(* Logix 5000 project; controller R1USB70001_CWRU_GRID_20120217 vendor 1 type 14 code 54 rev 19.11; software revision 19.01; part 3 of 3 *)
(* tags used below, declared in another part *)
   BAT_AC_VOLTAGE : REAL;
   BAT_AC_VOLTAGE_RAW : REAL;
   BAT_CHARGE_AC_CURRENT : REAL;
   BAT_CHARGE_AC_CURRENT_RAW : REAL;
   BAT_CHARGE_DC_CURRENT : REAL;
   BAT_CHARGE_DC_CURRENT_RAW : REAL;
   BAT_SRC_AC_CURRENT1 : REAL;
   BAT_SRC_AC_CURRENT1_RAW : REAL;
   BAT_SRC_AC_CURRENT2 : REAL;
   BAT_SRC_AC_CURRENT2_RAW : REAL;
   BAT_SRC_DC_CURRENT : REAL;
   BAT_SRC_DC_CURRENT_RAW : REAL;
   CAES_CHARGE_CURRENT : REAL;
   CAES_CHARGE_CURRENT_RAW : REAL;
   CAES_SRC_CURRENT : REAL;
   CAES_SRC_CURRENT_RAW : REAL;
   CAP_MAIN_CURRENT : REAL;
   CAP_MAIN_CURRENT_RAW : REAL;
   COM_TO_GRID_CURRENT : REAL;
   COM_TO_GRID_CURRENT_RAW : REAL;
   CURRENT_SCALE_HIGH : REAL;
   CURRENT_SCALE_LOW : REAL;
   IND_TO_GRID_CURRENT : REAL;
   IND_TO_GRID_CURRENT_RAW : REAL;
   MAINS_AC_VOLTAGE : REAL;
   MAINS_AC_VOLTAGE_RAW : REAL;
   RES_TO_GRID_CURRENT : REAL;
   RES_TO_GRID_CURRENT_RAW : REAL;
   SC_TO_BAT_CURRENT : REAL;
   SC_TO_BAT_CURRENT_RAW : REAL;
   SC_TO_COM_CURRENT : REAL;
   SC_TO_COM_CURRENT_RAW : REAL;
   SC_TO_GRID_CURRENT : REAL;
   SC_TO_GRID_CURRENT_RAW : REAL;
   SC_TO_IND_CURRENT : REAL;
   SC_TO_IND_CURRENT_RAW : REAL;
   SC_TO_RES_CURRENT : REAL;
   SC_TO_RES_CURRENT_RAW : REAL;
   SF_TO_BAT_CURRENT : REAL;
   SF_TO_BAT_CURRENT_RAW : REAL;
   SF_TO_COM_CURRENT : REAL;
   SF_TO_COM_CURRENT_RAW : REAL;
   SF_TO_GRID_CURRENT : REAL;
   SF_TO_GRID_CURRENT_RAW : REAL;
   SF_TO_IND_CURRENT : REAL;
   SF_TO_IND_CURRENT_RAW : REAL;
   SF_TO_RES_CURRENT : REAL;
   SF_TO_RES_CURRENT_RAW : REAL;
   VOLTAGE_SCALE : REAL;
   WF_TO_BAT_CURRENT : REAL;
   WF_TO_BAT_CURRENT_RAW : REAL;
   WF_TO_COM_CURRENT : REAL;
   WF_TO_COM_CURRENT_RAW : REAL;
   WF_TO_GRID_CURRENT : REAL;
   WF_TO_GRID_CURRENT_RAW : REAL;
   WF_TO_IND_CURRENT : REAL;
   WF_TO_IND_CURRENT_RAW : REAL;
   WF_TO_RES_CURRENT : REAL;
   WF_TO_RES_CURRENT_RAW : REAL;
   WT_TO_BAT_CURRENT : REAL;
   WT_TO_BAT_CURRENT_RAW : REAL;
   WT_TO_COM_CURRENT : REAL;
   WT_TO_COM_CURRENT_RAW : REAL;
   WT_TO_GRID_CURRENT : REAL;
   WT_TO_GRID_CURRENT_RAW : REAL;
   WT_TO_IND_CURRENT : REAL;
   WT_TO_IND_CURRENT_RAW : REAL;
   WT_TO_RES_CURRENT : REAL;
   WT_TO_RES_CURRENT_RAW : REAL;
   AP_GP_CH_ACAM : ALIAS FOR ACNR_GP_SC_N2:1:I.Ch1Data;
   AP_GP_SR_ACAM : ALIAS FOR ACNR_GP_SC_N2:1:I.Ch0Data;
   AP_GP_SR_ACVT : ALIAS FOR ACNR_GP_SC_N2:9:I.Ch1Data;
   BT_GP_L1_ACAM1 : ALIAS FOR ACNR_GP_SC_N2:1:I.Ch2Data;
   BT_GP_L1_ACAM2 : ALIAS FOR ACNR_GP_SC_N2:1:I.Ch3Data;
   BT_GP_L1_DCAM : ALIAS FOR ACNR_GP_SC_N2:2:I.Ch2Data;
   BT_GP_L2_ACAM1 : ALIAS FOR ACNR_GP_SC_N2:2:I.Ch0Data;
   BT_GP_L2_DCAM : ALIAS FOR ACNR_GP_SC_N2:2:I.Ch3Data;
   BT_GP_ML_ACVT : ALIAS FOR ACNR_GP_SC_N2:9:I.Ch2Data;
   CB_GP_ML_ACAM : ALIAS FOR ACNR_GP_SC_N2:9:I.Ch0Data;
   CL_GP_GD_ACAM : ALIAS FOR ACNR_GP_SC_N2:5:I.Ch2Data;
   CL_GP_SC_ACAM : ALIAS FOR ACNR_GP_SC_N2:4:I.Ch2Data;
   CL_GP_SF_ACAM : ALIAS FOR ACNR_GP_SC_N2:4:I.Ch3Data;
   CL_GP_WF_ACAM : ALIAS FOR ACNR_GP_SC_N2:5:I.Ch1Data;
   CL_GP_WT_ACAM : ALIAS FOR ACNR_GP_SC_N2:5:I.Ch0Data;
   Comment : DINT[2];
   IL_GP_GD_ACAM : ALIAS FOR ACNR_GP_SC_N2:6:I.Ch3Data;
   IL_GP_SC_ACAM : ALIAS FOR ACNR_GP_SC_N2:5:I.Ch3Data;
   IL_GP_SF_ACAM : ALIAS FOR ACNR_GP_SC_N2:6:I.Ch0Data;
   IL_GP_WF_ACAM : ALIAS FOR ACNR_GP_SC_N2:6:I.Ch2Data;
   IL_GP_WT_ACAM : ALIAS FOR ACNR_GP_SC_N2:6:I.Ch1Data;
   RL_GP_GD_ACAM : ALIAS FOR ACNR_GP_SC_N2:4:I.Ch1Data;
   RL_GP_SC_ACAM : ALIAS FOR ACNR_GP_SC_N2:3:I.Ch0Data;
   RL_GP_SF_ACAM : ALIAS FOR ACNR_GP_SC_N2:3:I.Ch1Data;
   RL_GP_WF_ACAM : ALIAS FOR ACNR_GP_SC_N2:4:I.Ch0Data;
   RL_GP_WT_ACAM : ALIAS FOR ACNR_GP_SC_N2:3:I.Ch2Data;
   SC_GP_BT_ACAM : ALIAS FOR ACNR_GP_SC_N2:8:I.Ch3Data;
   SC_GP_GD_ACAM : ALIAS FOR ACNR_GP_SC_N2:8:I.Ch2Data;
   SF_GP_BT_ACAM : ALIAS FOR ACNR_GP_SC_N2:8:I.Ch1Data;
   SF_GP_GD_ACAM : ALIAS FOR ACNR_GP_SC_N2:8:I.Ch0Data;
   WF_GP_BT_ACAM : ALIAS FOR ACNR_GP_SC_N2:7:I.Ch1Data;
   WF_GP_GD_ACAM : ALIAS FOR ACNR_GP_SC_N2:7:I.Ch0Data;
   WT_GP_BT_ACAM : ALIAS FOR ACNR_GP_SC_N2:7:I.Ch3Data;
   WT_GP_GD_ACAM : ALIAS FOR ACNR_GP_SC_N2:7:I.Ch2Data;
(* MainProgram, continued *)

ROUTINE IMPORT_DATA   (* ladder *)
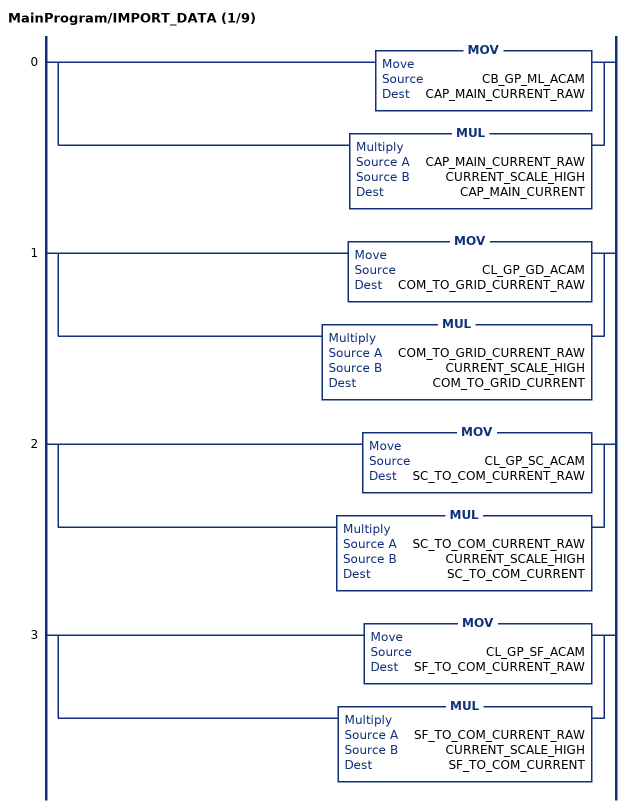
   0: [MOV(CB_GP_ML_ACAM,CAP_MAIN_CURRENT_RAW) ,MUL(CAP_MAIN_CURRENT_RAW,CURRENT_SCALE_HIGH,CAP_MAIN_CURRENT) ];
   1: [MOV(CL_GP_GD_ACAM,COM_TO_GRID_CURRENT_RAW) ,MUL(COM_TO_GRID_CURRENT_RAW,CURRENT_SCALE_HIGH,COM_TO_GRID_CURRENT) ];
   2: [MOV(CL_GP_SC_ACAM,SC_TO_COM_CURRENT_RAW) ,MUL(SC_TO_COM_CURRENT_RAW,CURRENT_SCALE_HIGH,SC_TO_COM_CURRENT) ];
   3: [MOV(CL_GP_SF_ACAM,SF_TO_COM_CURRENT_RAW) ,MUL(SF_TO_COM_CURRENT_RAW,CURRENT_SCALE_HIGH,SF_TO_COM_CURRENT) ];
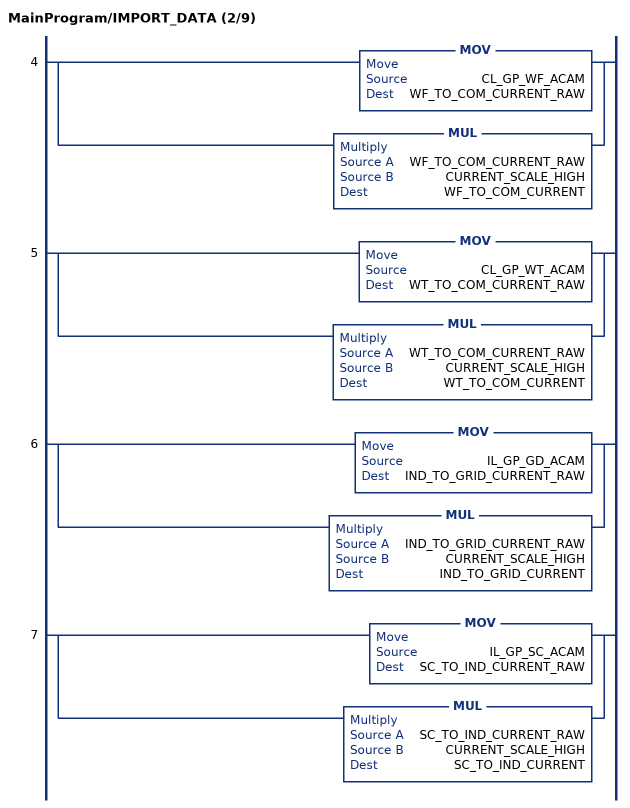
   4: [MOV(CL_GP_WF_ACAM,WF_TO_COM_CURRENT_RAW) ,MUL(WF_TO_COM_CURRENT_RAW,CURRENT_SCALE_HIGH,WF_TO_COM_CURRENT) ];
   5: [MOV(CL_GP_WT_ACAM,WT_TO_COM_CURRENT_RAW) ,MUL(WT_TO_COM_CURRENT_RAW,CURRENT_SCALE_HIGH,WT_TO_COM_CURRENT) ];
   6: [MOV(IL_GP_GD_ACAM,IND_TO_GRID_CURRENT_RAW) ,MUL(IND_TO_GRID_CURRENT_RAW,CURRENT_SCALE_HIGH,IND_TO_GRID_CURRENT) ];
   7: [MOV(IL_GP_SC_ACAM,SC_TO_IND_CURRENT_RAW) ,MUL(SC_TO_IND_CURRENT_RAW,CURRENT_SCALE_HIGH,SC_TO_IND_CURRENT) ];
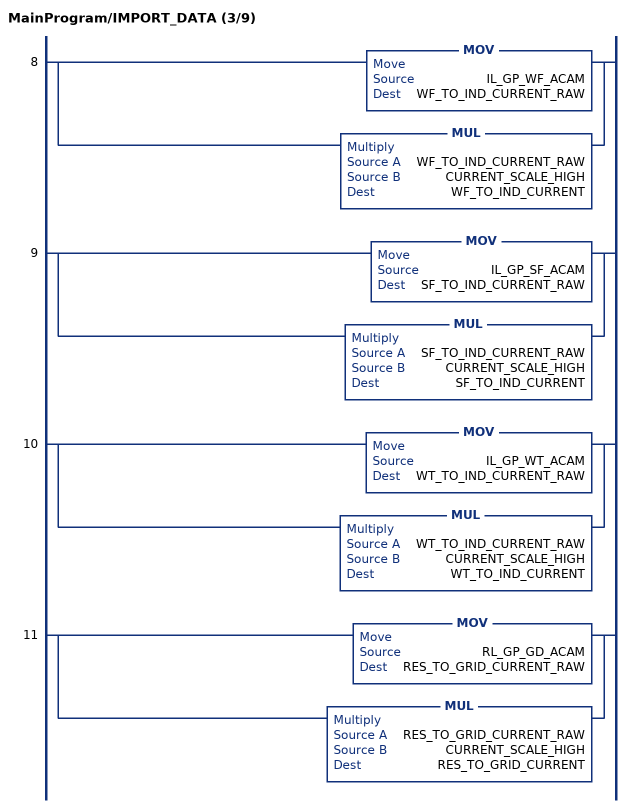
   8: [MOV(IL_GP_WF_ACAM,WF_TO_IND_CURRENT_RAW) ,MUL(WF_TO_IND_CURRENT_RAW,CURRENT_SCALE_HIGH,WF_TO_IND_CURRENT) ];
   9: [MOV(IL_GP_SF_ACAM,SF_TO_IND_CURRENT_RAW) ,MUL(SF_TO_IND_CURRENT_RAW,CURRENT_SCALE_HIGH,SF_TO_IND_CURRENT) ];
   10: [MOV(IL_GP_WT_ACAM,WT_TO_IND_CURRENT_RAW) ,MUL(WT_TO_IND_CURRENT_RAW,CURRENT_SCALE_HIGH,WT_TO_IND_CURRENT) ];
   11: [MOV(RL_GP_GD_ACAM,RES_TO_GRID_CURRENT_RAW) ,MUL(RES_TO_GRID_CURRENT_RAW,CURRENT_SCALE_HIGH,RES_TO_GRID_CURRENT) ];
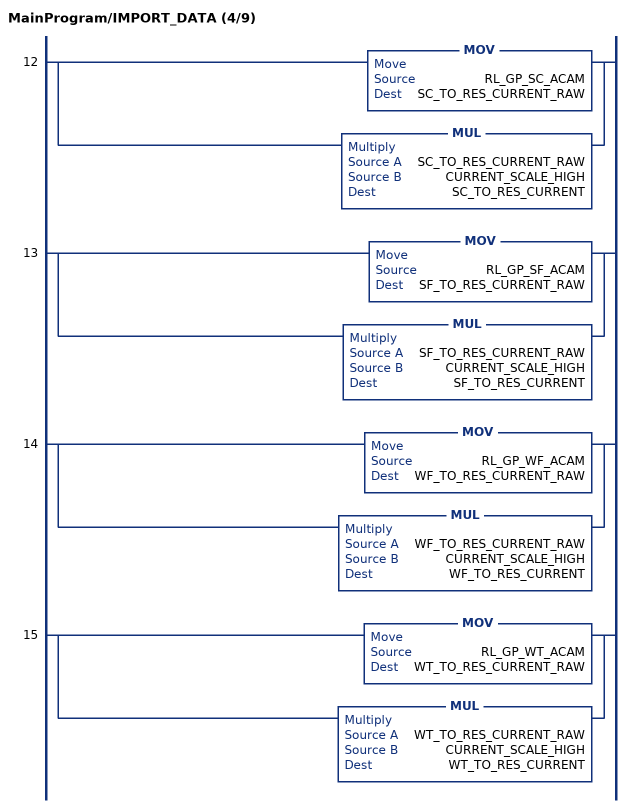
   12: [MOV(RL_GP_SC_ACAM,SC_TO_RES_CURRENT_RAW) ,MUL(SC_TO_RES_CURRENT_RAW,CURRENT_SCALE_HIGH,SC_TO_RES_CURRENT) ];
   13: [MOV(RL_GP_SF_ACAM,SF_TO_RES_CURRENT_RAW) ,MUL(SF_TO_RES_CURRENT_RAW,CURRENT_SCALE_HIGH,SF_TO_RES_CURRENT) ];
   14: [MOV(RL_GP_WF_ACAM,WF_TO_RES_CURRENT_RAW) ,MUL(WF_TO_RES_CURRENT_RAW,CURRENT_SCALE_HIGH,WF_TO_RES_CURRENT) ];
   15: [MOV(RL_GP_WT_ACAM,WT_TO_RES_CURRENT_RAW) ,MUL(WT_TO_RES_CURRENT_RAW,CURRENT_SCALE_HIGH,WT_TO_RES_CURRENT) ];
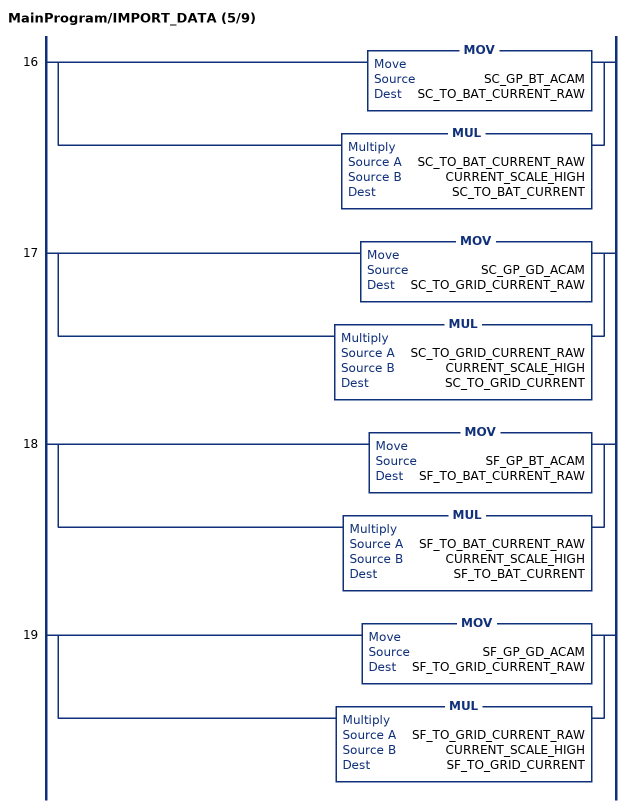
   16: [MOV(SC_GP_BT_ACAM,SC_TO_BAT_CURRENT_RAW) ,MUL(SC_TO_BAT_CURRENT_RAW,CURRENT_SCALE_HIGH,SC_TO_BAT_CURRENT) ];
   17: [MOV(SC_GP_GD_ACAM,SC_TO_GRID_CURRENT_RAW) ,MUL(SC_TO_GRID_CURRENT_RAW,CURRENT_SCALE_HIGH,SC_TO_GRID_CURRENT) ];
   18: [MOV(SF_GP_BT_ACAM,SF_TO_BAT_CURRENT_RAW) ,MUL(SF_TO_BAT_CURRENT_RAW,CURRENT_SCALE_HIGH,SF_TO_BAT_CURRENT) ];
   19: [MOV(SF_GP_GD_ACAM,SF_TO_GRID_CURRENT_RAW) ,MUL(SF_TO_GRID_CURRENT_RAW,CURRENT_SCALE_HIGH,SF_TO_GRID_CURRENT) ];
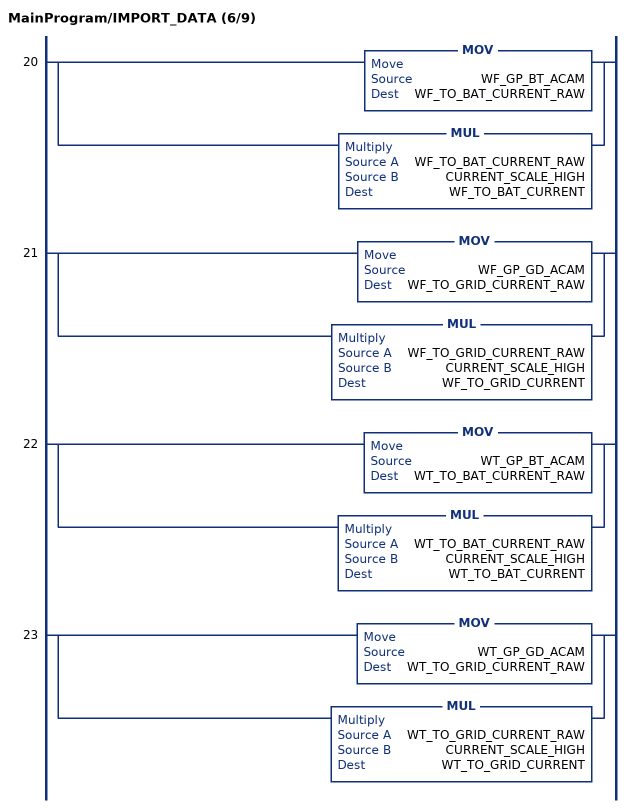
   20: [MOV(WF_GP_BT_ACAM,WF_TO_BAT_CURRENT_RAW) ,MUL(WF_TO_BAT_CURRENT_RAW,CURRENT_SCALE_HIGH,WF_TO_BAT_CURRENT) ];
   21: [MOV(WF_GP_GD_ACAM,WF_TO_GRID_CURRENT_RAW) ,MUL(WF_TO_GRID_CURRENT_RAW,CURRENT_SCALE_HIGH,WF_TO_GRID_CURRENT) ];
   22: [MOV(WT_GP_BT_ACAM,WT_TO_BAT_CURRENT_RAW) ,MUL(WT_TO_BAT_CURRENT_RAW,CURRENT_SCALE_HIGH,WT_TO_BAT_CURRENT) ];
   23: [MOV(WT_GP_GD_ACAM,WT_TO_GRID_CURRENT_RAW) ,MUL(WT_TO_GRID_CURRENT_RAW,CURRENT_SCALE_HIGH,WT_TO_GRID_CURRENT) ];
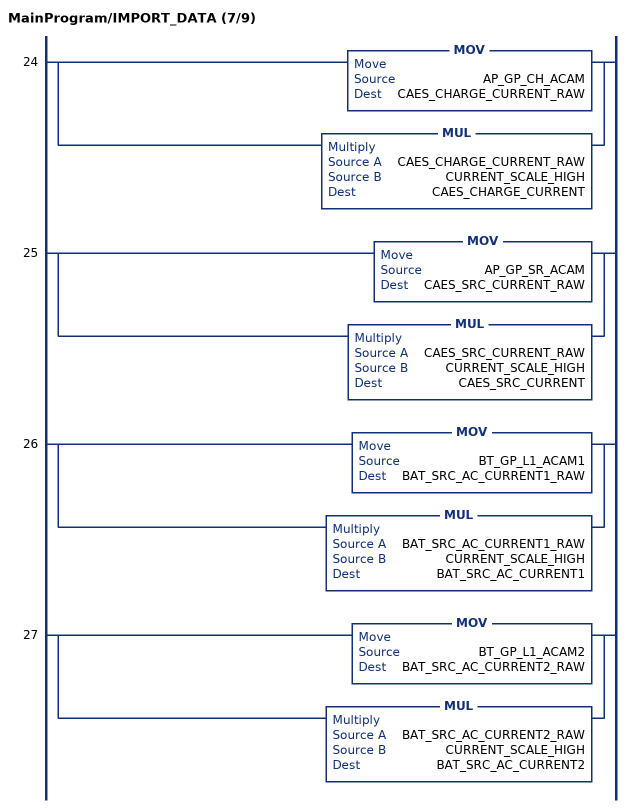
   24: [MOV(AP_GP_CH_ACAM,CAES_CHARGE_CURRENT_RAW) ,MUL(CAES_CHARGE_CURRENT_RAW,CURRENT_SCALE_HIGH,CAES_CHARGE_CURRENT) ];
   25: [MOV(AP_GP_SR_ACAM,CAES_SRC_CURRENT_RAW) ,MUL(CAES_SRC_CURRENT_RAW,CURRENT_SCALE_HIGH,CAES_SRC_CURRENT) ];
   26: [MOV(BT_GP_L1_ACAM1,BAT_SRC_AC_CURRENT1_RAW) ,MUL(BAT_SRC_AC_CURRENT1_RAW,CURRENT_SCALE_HIGH,BAT_SRC_AC_CURRENT1) ];
   27: [MOV(BT_GP_L1_ACAM2,BAT_SRC_AC_CURRENT2_RAW) ,MUL(BAT_SRC_AC_CURRENT2_RAW,CURRENT_SCALE_HIGH,BAT_SRC_AC_CURRENT2) ];
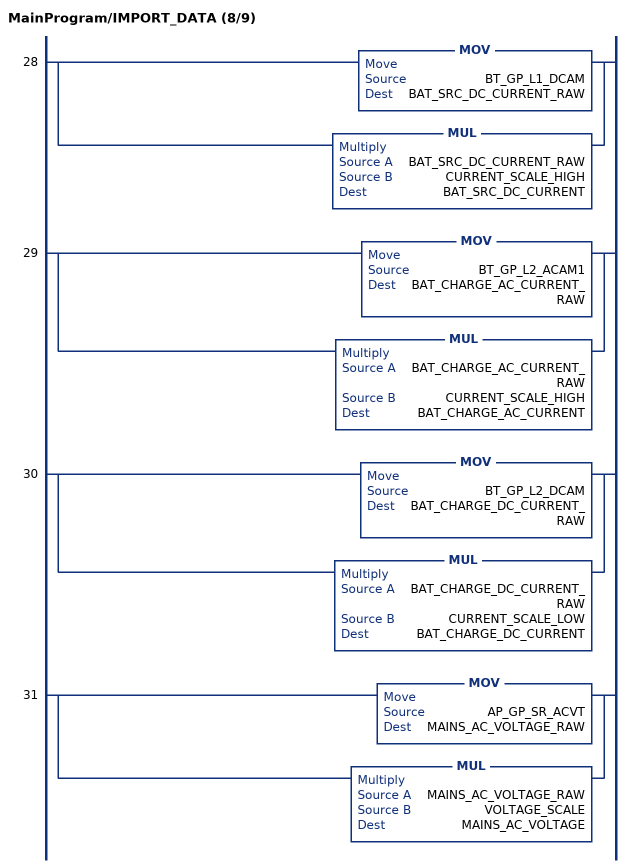
   28: [MOV(BT_GP_L1_DCAM,BAT_SRC_DC_CURRENT_RAW) ,MUL(BAT_SRC_DC_CURRENT_RAW,CURRENT_SCALE_HIGH,BAT_SRC_DC_CURRENT) ];
   29: [MOV(BT_GP_L2_ACAM1,BAT_CHARGE_AC_CURRENT_RAW) ,MUL(BAT_CHARGE_AC_CURRENT_RAW,CURRENT_SCALE_HIGH,BAT_CHARGE_AC_CURRENT) ];
   30: [MOV(BT_GP_L2_DCAM,BAT_CHARGE_DC_CURRENT_RAW) ,MUL(BAT_CHARGE_DC_CURRENT_RAW,CURRENT_SCALE_LOW,BAT_CHARGE_DC_CURRENT) ];
   31: [MOV(AP_GP_SR_ACVT,MAINS_AC_VOLTAGE_RAW) ,MUL(MAINS_AC_VOLTAGE_RAW,VOLTAGE_SCALE,MAINS_AC_VOLTAGE) ];
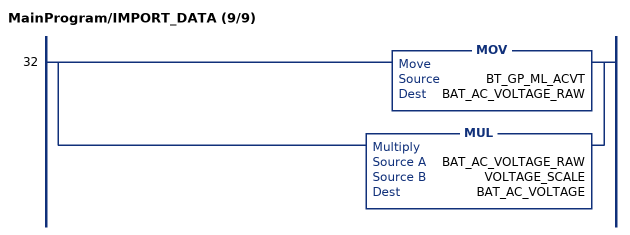
   32: [MOV(BT_GP_ML_ACVT,BAT_AC_VOLTAGE_RAW) ,MUL(BAT_AC_VOLTAGE_RAW,VOLTAGE_SCALE,BAT_AC_VOLTAGE) ];
END_ROUTINE

ROUTINE MainRoutine   (* ladder *)
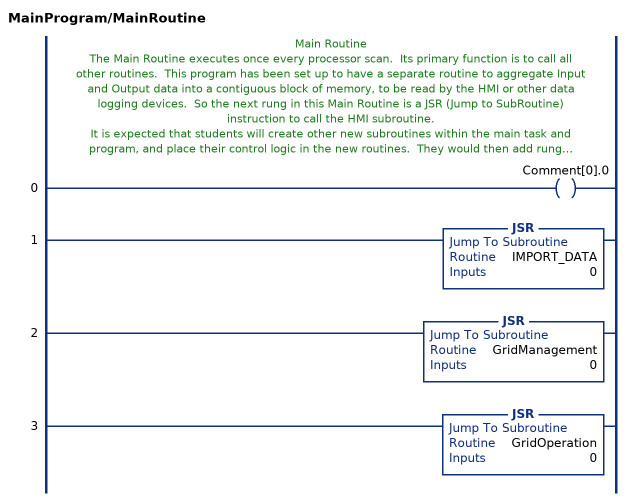
   // Main Routine
   // The Main Routine executes once every processor scan.  Its primary function is to call all other routines.  This program has been set up to have a separate routine to aggregate Input and Output data into a contiguous block of memory, to be read by the HMI or other data logging devices.  So the next rung in this Main Routine is a JSR (Jump to SubRoutine) instruction to call the HMI subroutine.
   // It is expected that students will create other new subroutines within the main task and program, and place their control logic in the new routines.  They would then add rungs within this Main Routine to call the new subroutines that contain their logic.
   0: OTE(Comment[0].0);
   1: JSR(IMPORT_DATA,0);
   2: JSR(GridManagement,0);
   3: JSR(GridOperation,0);
END_ROUTINE
END_PROGRAM
